// Mitsubishi GX Works2 project: continuous_sequence   PLC: Q03UDV

PROGRAM MAIN
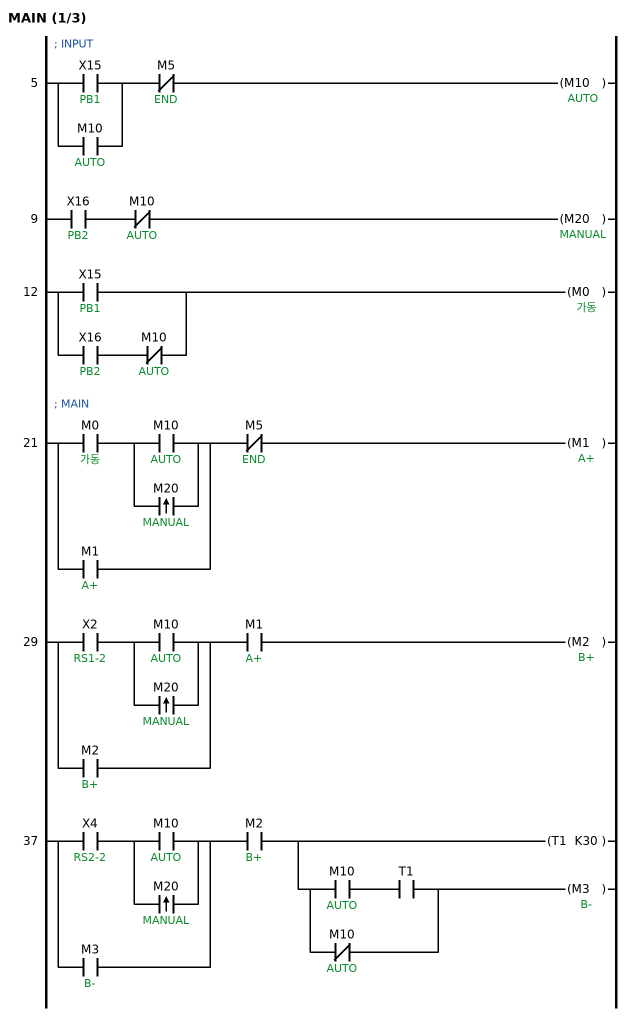
; INPUT
5     LD      X15  ; PB1
      OR      M10  ; AUTO
      ANI     M5  ; END
      OUT     M10  ; AUTO
9     LD      X16  ; PB2
      ANI     M10  ; AUTO
      OUT     M20  ; MANUAL
12    LD      X15  ; PB1
      LD      X16  ; PB2
      ANI     M10  ; AUTO
      ORB
      OUT     M0  ; 가동
; MAIN
21    LD      M0  ; 가동
      LD      M10  ; AUTO
      ORP     M20  ; MANUAL
      ANB
      OR      M1  ; A+
      ANI     M5  ; END
      OUT     M1  ; A+
29    LD      X2  ; RS1-2
      LD      M10  ; AUTO
      ORP     M20  ; MANUAL
      ANB
      OR      M2  ; B+
      AND     M1  ; A+
      OUT     M2  ; B+
37    LD      X4  ; RS2-2
      LD      M10  ; AUTO
      ORP     M20  ; MANUAL
      ANB
      OR      M3  ; B-
      AND     M2  ; B+
      OUT     T1 K30
      LD      M10  ; AUTO
      AND     T1
      ORI     M10  ; AUTO
      ANB
      OUT     M3  ; B-
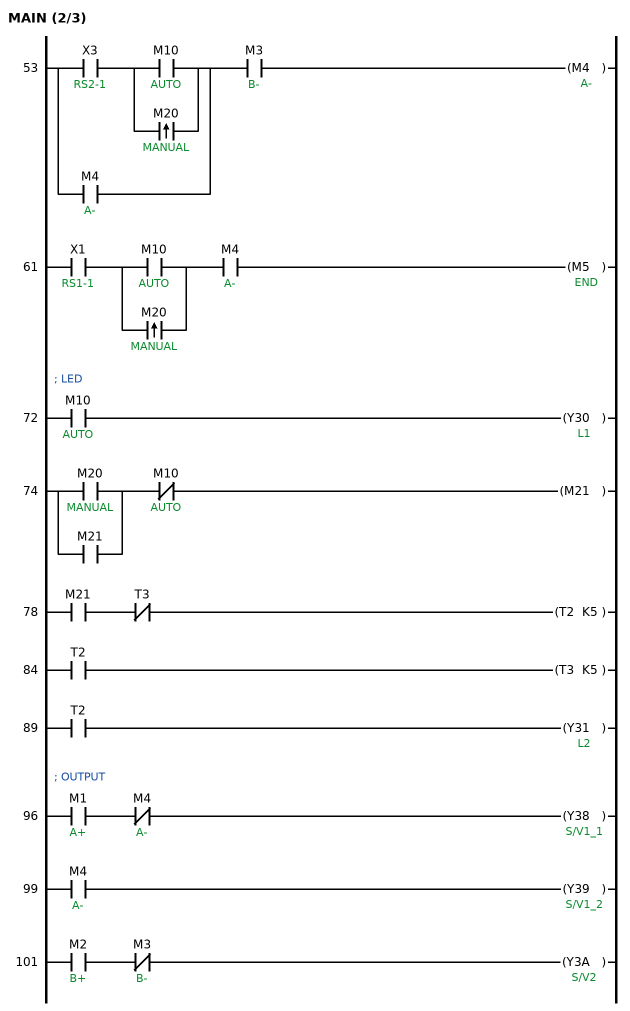
53    LD      X3  ; RS2-1
      LD      M10  ; AUTO
      ORP     M20  ; MANUAL
      ANB
      OR      M4  ; A-
      AND     M3  ; B-
      OUT     M4  ; A-
61    LD      X1  ; RS1-1
      LD      M10  ; AUTO
      ORP     M20  ; MANUAL
      ANB
      AND     M4  ; A-
      OUT     M5  ; END
; LED
72    LD      M10  ; AUTO
      OUT     Y30  ; L1
74    LD      M20  ; MANUAL
      OR      M21
      ANI     M10  ; AUTO
      OUT     M21
78    LD      M21
      ANI     T3
      OUT     T2 K5
84    LD      T2
      OUT     T3 K5
89    LD      T2
      OUT     Y31  ; L2
; OUTPUT
96    LD      M1  ; A+
      ANI     M4  ; A-
      OUT     Y38  ; S/V1_1
99    LD      M4  ; A-
      OUT     Y39  ; S/V1_2
101   LD      M2  ; B+
      ANI     M3  ; B-
      OUT     Y3A  ; S/V2
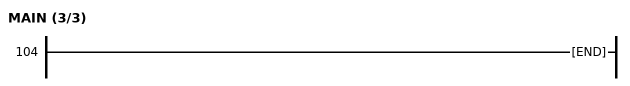
104   END
END_PROGRAM

// device comments not shown above
X17  ; PB3
X18  ; PB4
X19  ; PB5
X1A  ; PB6
X1B  ; PB7
X1C  ; PB8
M14  ; B+
M15  ; B-
M22  ; B-
M24  ; A+
M25  ; A-
Y32  ; L3
Y33  ; L4
Y34  ; L5
Y35  ; L6
Y36  ; L7
Y37  ; Buzzer
Y3B  ; S/V3
